// TIA Portal project "timers" (V15)

(* hardware
DEVICE "S7-1200 station_1"  S7-1200 Station
   slot 0: "Rack_0"  S7-1200 Rack  Rack  V1.0
   slot 1: "PLC_1"  CPU 1212C DC/DC/DC  6ES7 212-1AE40-0XB0  V4.2
*)

// ===== PLC "PLC_1"  CPU 1212C DC/DC/DC =====

VAR_GLOBAL   // PLC tag table "Default tag table"
   "sw1" AT %M0.1 : Bool;
   "Tag_1" AT %Q0.1 : Bool;
   "Tag_2" AT %Q0.2 : Bool;
   "Tag_3" AT %M1.1 : Bool;
   "Tag_4" AT %Q1.1 : Bool;
   "Tag_5" AT %Q1.2 : Bool;
   "Tag_6" AT %Q1.3 : Bool;
   "Tag_7" AT %M1.2 : Bool;
   "Tag_8" AT %Q2.1 : Bool;
   "low sensor" AT %M3.1 : Bool;
   "heater" AT %Q3.1 : Bool;
   "high sensor" AT %M30.2 : Bool;
   "cooler" AT %Q3.2 : Bool;
   "Tag_9" AT %M4.0 : Bool;
   "Tag_10" AT %Q4.0 : Bool;
   "Tag_11" AT %M6.1 : Bool;
   "Tag_12" AT %Q6.1 : Bool;
   "Tag_13" AT %M7.1 : Bool;
   "Tag_14" AT %Q7.1 : Bool;
   "Tag_15" AT %M8.1 : Bool;
   "FILLING" AT %Q8.1 : Bool;
   "AGITATION" AT %Q8.2 : Bool;
   "DRAIN" AT %Q8.3 : Bool;
   "SPIN" AT %Q8.4 : Bool;
   "ALARAM" AT %Q8.5 : Bool;
   "SW" AT %M9.1 : Bool;
   "PUMP" AT %Q9.1 : Bool;
   "VALVE1" AT %Q9.2 : Bool;
   "VALVE3" AT %Q9.3 : Bool;
   "MIXTURE" AT %Q9.4 : Bool;
   "PUMP2" AT %Q9.5 : Bool;
   "DRAIN(1)" AT %Q9.6 : Bool;
   "Tag_16" AT %M2.5 : Bool;
   "Tag_17" AT %M2.6 : Bool;
   "Tag_18" AT %Q2.5 : Bool;
   "drain(2)" AT %Q2.6 : Bool;
   "Tag_19" AT %Q6.5 : Bool;
   "tank" AT %Q0.6 : Bool;
END_VAR

// folder: System blocks/Program resources

DATA_BLOCK "IEC_Timer_0_DB"   // DB1
{ S7_Optimized_Access := 'TRUE' }
AUTHOR : Simatic
FAMILY : IEC
NAME : IEC_TMR
VERSION : 1.0
// stored: InstanceOfName IEC_TIMER
"IEC_TIMER"
BEGIN
END_DATA_BLOCK

DATA_BLOCK "IEC_Timer_0_DB_1"   // DB2
{ S7_Optimized_Access := 'TRUE' }
AUTHOR : Simatic
FAMILY : IEC
NAME : IEC_TMR
VERSION : 1.0
// stored: InstanceOfName IEC_TIMER
"IEC_TIMER"
BEGIN
END_DATA_BLOCK

DATA_BLOCK "IEC_Timer_0_DB_2"   // DB3
{ S7_Optimized_Access := 'TRUE' }
AUTHOR : Simatic
FAMILY : IEC
NAME : IEC_TMR
VERSION : 1.0
// stored: InstanceOfName IEC_TIMER
"IEC_TIMER"
BEGIN
END_DATA_BLOCK

DATA_BLOCK "IEC_Timer_0_DB_3"   // DB4
{ S7_Optimized_Access := 'TRUE' }
AUTHOR : Simatic
FAMILY : IEC
NAME : IEC_TMR
VERSION : 1.0
// stored: InstanceOfName IEC_TIMER
"IEC_TIMER"
BEGIN
END_DATA_BLOCK

DATA_BLOCK "IEC_Timer_0_DB_4"   // DB5
{ S7_Optimized_Access := 'TRUE' }
AUTHOR : Simatic
FAMILY : IEC
NAME : IEC_TMR
VERSION : 1.0
// stored: InstanceOfName IEC_TIMER
"IEC_TIMER"
BEGIN
END_DATA_BLOCK

DATA_BLOCK "IEC_Timer_0_DB_5"   // DB6
{ S7_Optimized_Access := 'TRUE' }
AUTHOR : Simatic
FAMILY : IEC
NAME : IEC_TMR
VERSION : 1.0
// stored: InstanceOfName IEC_TIMER
"IEC_TIMER"
BEGIN
END_DATA_BLOCK

DATA_BLOCK "IEC_Timer_0_DB_6"   // DB7
{ S7_Optimized_Access := 'TRUE' }
AUTHOR : Simatic
FAMILY : IEC
NAME : IEC_TMR
VERSION : 1.0
// stored: InstanceOfName IEC_TIMER
"IEC_TIMER"
BEGIN
END_DATA_BLOCK

DATA_BLOCK "IEC_Timer_0_DB_7"   // DB8
{ S7_Optimized_Access := 'TRUE' }
AUTHOR : Simatic
FAMILY : IEC
NAME : IEC_TMR
VERSION : 1.0
// stored: InstanceOfName IEC_TIMER
"IEC_TIMER"
BEGIN
END_DATA_BLOCK

DATA_BLOCK "IEC_Timer_0_DB_8"   // DB9
{ S7_Optimized_Access := 'TRUE' }
AUTHOR : Simatic
FAMILY : IEC
NAME : IEC_TMR
VERSION : 1.0
// stored: InstanceOfName IEC_TIMER
"IEC_TIMER"
BEGIN
END_DATA_BLOCK

DATA_BLOCK "IEC_Timer_0_DB_9"   // DB10
{ S7_Optimized_Access := 'TRUE' }
AUTHOR : Simatic
FAMILY : IEC
NAME : IEC_TMR
VERSION : 1.0
// stored: InstanceOfName IEC_TIMER
"IEC_TIMER"
BEGIN
END_DATA_BLOCK

DATA_BLOCK "IEC_Timer_0_DB_10"   // DB11
{ S7_Optimized_Access := 'TRUE' }
AUTHOR : Simatic
FAMILY : IEC
NAME : IEC_TMR
VERSION : 1.0
// stored: InstanceOfName IEC_TIMER
"IEC_TIMER"
BEGIN
END_DATA_BLOCK

DATA_BLOCK "IEC_Timer_0_DB_11"   // DB12
{ S7_Optimized_Access := 'TRUE' }
AUTHOR : Simatic
FAMILY : IEC
NAME : IEC_TMR
VERSION : 1.0
// stored: InstanceOfName IEC_TIMER
"IEC_TIMER"
BEGIN
END_DATA_BLOCK

DATA_BLOCK "IEC_Timer_0_DB_12"   // DB13
{ S7_Optimized_Access := 'TRUE' }
AUTHOR : Simatic
FAMILY : IEC
NAME : IEC_TMR
VERSION : 1.0
// stored: InstanceOfName IEC_TIMER
"IEC_TIMER"
BEGIN
END_DATA_BLOCK

DATA_BLOCK "IEC_Timer_0_DB_13"   // DB14
{ S7_Optimized_Access := 'TRUE' }
AUTHOR : Simatic
FAMILY : IEC
NAME : IEC_TMR
VERSION : 1.0
// stored: InstanceOfName IEC_TIMER
"IEC_TIMER"
BEGIN
END_DATA_BLOCK

DATA_BLOCK "IEC_Timer_0_DB_14"   // DB15
{ S7_Optimized_Access := 'TRUE' }
AUTHOR : Simatic
FAMILY : IEC
NAME : IEC_TMR
VERSION : 1.0
// stored: InstanceOfName IEC_TIMER
"IEC_TIMER"
BEGIN
END_DATA_BLOCK

DATA_BLOCK "IEC_Timer_0_DB_15"   // DB16
{ S7_Optimized_Access := 'TRUE' }
AUTHOR : Simatic
FAMILY : IEC
NAME : IEC_TMR
VERSION : 1.0
// stored: InstanceOfName IEC_TIMER
"IEC_TIMER"
BEGIN
END_DATA_BLOCK

DATA_BLOCK "IEC_Timer_0_DB_16"   // DB17
{ S7_Optimized_Access := 'TRUE' }
AUTHOR : Simatic
FAMILY : IEC
NAME : IEC_TMR
VERSION : 1.0
// stored: InstanceOfName IEC_TIMER
"IEC_TIMER"
BEGIN
END_DATA_BLOCK

DATA_BLOCK "IEC_Timer_0_DB_17"   // DB18
{ S7_Optimized_Access := 'TRUE' }
AUTHOR : Simatic
FAMILY : IEC
NAME : IEC_TMR
VERSION : 1.0
// stored: InstanceOfName IEC_TIMER
"IEC_TIMER"
BEGIN
END_DATA_BLOCK

DATA_BLOCK "IEC_Timer_0_DB_18"   // DB19
{ S7_Optimized_Access := 'TRUE' }
AUTHOR : Simatic
FAMILY : IEC
NAME : IEC_TMR
VERSION : 1.0
// stored: InstanceOfName IEC_TIMER
"IEC_TIMER"
BEGIN
END_DATA_BLOCK

DATA_BLOCK "IEC_Timer_0_DB_19"   // DB20
{ S7_Optimized_Access := 'TRUE' }
AUTHOR : Simatic
FAMILY : IEC
NAME : IEC_TMR
VERSION : 1.0
// stored: InstanceOfName IEC_TIMER
"IEC_TIMER"
BEGIN
END_DATA_BLOCK

DATA_BLOCK "IEC_Timer_0_DB_26"   // DB27
{ S7_Optimized_Access := 'TRUE' }
AUTHOR : Simatic
FAMILY : IEC
NAME : IEC_TMR
VERSION : 1.0
// stored: InstanceOfName IEC_TIMER
"IEC_TIMER"
BEGIN
END_DATA_BLOCK

// folder: (top level)

ORGANIZATION_BLOCK "Main"   // OB1, LAD, ProgramCycle
TITLE = "Main Program Sweep (Cycle)"
{ S7_Optimized_Access := 'TRUE' }
VERSION : 0.1
   VAR_INPUT
      Initial_Call : Bool;   // Initial call of this OB
      Remanence : Bool;   // =True, if remanent data are available
   END_VAR
BEGIN

REGION Network 1
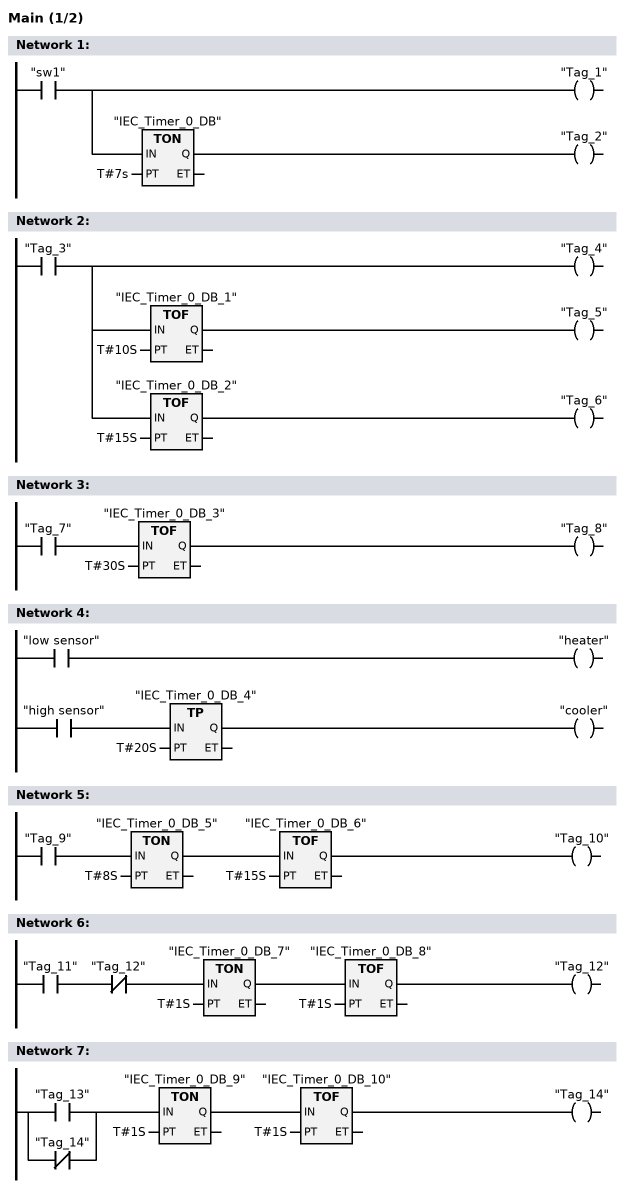
   "Tag_1" := "sw1";
   "IEC_Timer_0_DB".TON(IN := "sw1", PT := T#7s);
   "Tag_2" := "IEC_Timer_0_DB".Q;
END_REGION

REGION Network 2
   "Tag_4" := "Tag_3";
   "IEC_Timer_0_DB_1".TOF(IN := "Tag_3", PT := T#10S);
   "Tag_5" := "IEC_Timer_0_DB_1".Q;
   "IEC_Timer_0_DB_2".TOF(IN := "Tag_3", PT := T#15S);
   "Tag_6" := "IEC_Timer_0_DB_2".Q;
END_REGION

REGION Network 3
   "IEC_Timer_0_DB_3".TOF(IN := "Tag_7", PT := T#30S);
   "Tag_8" := "IEC_Timer_0_DB_3".Q;
END_REGION

REGION Network 4
   "heater" := "low sensor";
   "IEC_Timer_0_DB_4".TP(IN := "high sensor", PT := T#20S);
   "cooler" := "IEC_Timer_0_DB_4".Q;
END_REGION

REGION Network 5
   "IEC_Timer_0_DB_5".TON(IN := "Tag_9", PT := T#8S);
   "IEC_Timer_0_DB_6".TOF(IN := "IEC_Timer_0_DB_5".Q, PT := T#15S);
   "Tag_10" := "IEC_Timer_0_DB_6".Q;
END_REGION

REGION Network 6
   "IEC_Timer_0_DB_7".TON(IN := "Tag_11" AND NOT "Tag_12", PT := T#1S);
   "IEC_Timer_0_DB_8".TOF(IN := "IEC_Timer_0_DB_7".Q, PT := T#1S);
   "Tag_12" := "IEC_Timer_0_DB_8".Q;
END_REGION

REGION Network 7
   "IEC_Timer_0_DB_9".TON(IN := "Tag_13" OR NOT "Tag_14", PT := T#1S);
   "IEC_Timer_0_DB_10".TOF(IN := "IEC_Timer_0_DB_9".Q, PT := T#1S);
   "Tag_14" := "IEC_Timer_0_DB_10".Q;
END_REGION

REGION Network 8
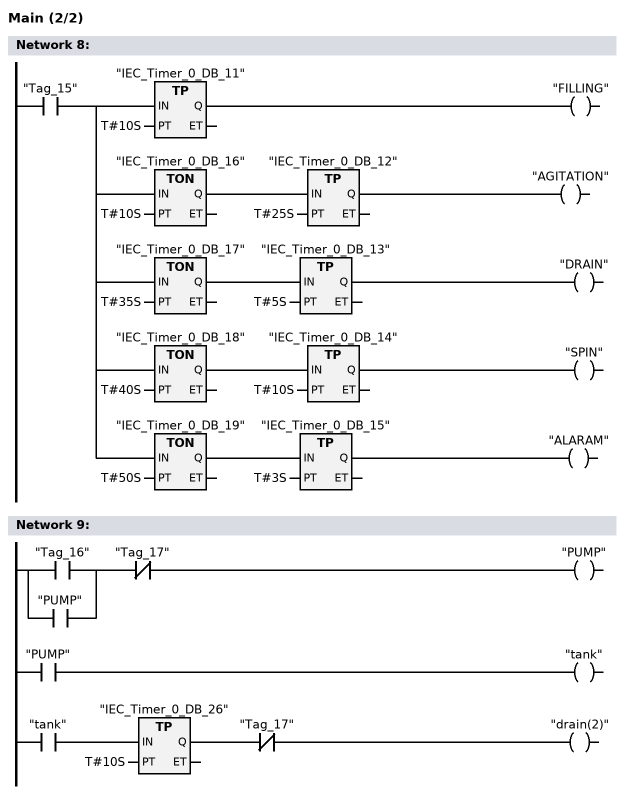
   "IEC_Timer_0_DB_11".TP(IN := "Tag_15", PT := T#10S);
   "FILLING" := "IEC_Timer_0_DB_11".Q;
   "IEC_Timer_0_DB_16".TON(IN := "Tag_15", PT := T#10S);
   "IEC_Timer_0_DB_12".TP(IN := "IEC_Timer_0_DB_16".Q, PT := T#25S);
   "AGITATION" := "IEC_Timer_0_DB_12".Q;
   "IEC_Timer_0_DB_17".TON(IN := "Tag_15", PT := T#35S);
   "IEC_Timer_0_DB_13".TP(IN := "IEC_Timer_0_DB_17".Q, PT := T#5S);
   "DRAIN" := "IEC_Timer_0_DB_13".Q;
   "IEC_Timer_0_DB_18".TON(IN := "Tag_15", PT := T#40S);
   "IEC_Timer_0_DB_14".TP(IN := "IEC_Timer_0_DB_18".Q, PT := T#10S);
   "SPIN" := "IEC_Timer_0_DB_14".Q;
   "IEC_Timer_0_DB_19".TON(IN := "Tag_15", PT := T#50S);
   "IEC_Timer_0_DB_15".TP(IN := "IEC_Timer_0_DB_19".Q, PT := T#3S);
   "ALARAM" := "IEC_Timer_0_DB_15".Q;
END_REGION

REGION Network 9
   "PUMP" := ("Tag_16" OR "PUMP") AND NOT "Tag_17";
   "tank" := "PUMP";
   "IEC_Timer_0_DB_26".TP(IN := "tank", PT := T#10S);
   "drain(2)" := "IEC_Timer_0_DB_26".Q AND NOT "Tag_17";
END_REGION
END_ORGANIZATION_BLOCK